TYPE Basic_Status_typ : 	
	STRUCT 
		Done : BOOL;
		Busy : BOOL;
		CommandAborted : BOOL;
		Active : BOOL ;
	END_STRUCT
END_TYPE

(* stored: Version 1.1.0.1, ProductVersion 3.1.4024.3
   DUT Basic_Status_typ: Id {71c8ba6d-6a67-0e5b-1adc-467befac9e46} *)
